(* IEC 61131-3 sources: industrial-ai-agent/projects/EXAMPLE_conveyor/program, 4 files *)

(* ---- 00_DUTs.st ---- *)
// ============================================================
// DUT (Data Unit Types) — Numaralandirmalar
// Proje: EXAMPLE_Conveyor_Line1
// Aciklama: Bolge mod ve durum makinesi tipleri
// ============================================================

// Bolge calisma modu
TYPE E_ZoneMode :
(
    MODE_MANUAL := 0,   // Operator buton ile kontrol
    MODE_AUTO   := 1    // Otomatik sira / fotosel ile
) := MODE_MANUAL;
END_TYPE

// Bolge durum makinesi
TYPE E_ZoneState :
(
    STATE_IDLE     := 0,    // Bekliyor, motor kapali
    STATE_STARTING := 1,    // Baslatma gecisi
    STATE_RUNNING  := 2,    // Calisiyor
    STATE_STOPPING := 3,    // Durdurma gecisi
    STATE_JAMMED   := 4,    // Sikisma - reset bekliyor
    STATE_FAULT    := 5     // Hata (hiz/diger) - reset bekliyor
) := STATE_IDLE;
END_TYPE

(* ---- 01_GVL_IO.st ---- *)
// ============================================================
// GVL_IO — Fiziksel Giris/Cikis degiskenleri
// Adresler io_list.csv ile BIREBIR tutarli olmalidir.
// Tek-yazar disiplini: cikislari yalniz ilgili PRG yazar.
// ============================================================
{attribute 'qualified_only'}
VAR_GLOBAL
    // --- Dijital Girisler (DI) ---
    ZN1_SEL_01_Auto    AT %IX0.0 : BOOL;   // Bolge 1 Oto/Manuel
    ZN1_PBS_01_Start   AT %IX0.1 : BOOL;
    ZN1_PBS_01_Stop    AT %IX0.2 : BOOL;   // NC: 1=normal, 0=basili
    ZN1_JAM_01_Sensor  AT %IX0.3 : BOOL;
    ZN1_PEY_01_Present AT %IX0.4 : BOOL;
    ZN2_SEL_02_Auto    AT %IX0.5 : BOOL;
    ZN2_PBS_02_Start   AT %IX0.6 : BOOL;
    ZN2_PBS_02_Stop    AT %IX0.7 : BOOL;
    ZN2_JAM_02_Sensor  AT %IX1.0 : BOOL;
    ZN2_PEY_02_Present AT %IX1.1 : BOOL;
    ZN3_SEL_03_Auto    AT %IX1.2 : BOOL;
    ZN3_PBS_03_Start   AT %IX1.3 : BOOL;
    ZN3_PBS_03_Stop    AT %IX1.4 : BOOL;
    ZN3_JAM_03_Sensor  AT %IX1.5 : BOOL;
    ZN3_PEY_03_Present AT %IX1.6 : BOOL;
    PLT_EST_01_OK      AT %IX1.7 : BOOL;   // Acil durdurma zinciri saglam (NC=1)
    PLT_RST_01_PB      AT %IX2.0 : BOOL;   // Reset / hata kabul
    PLT_PMT_01_Run     AT %IX2.1 : BOOL;   // Calistirma izni (NC)

    // --- Dijital Cikislar (DO) ---
    ZN1_MTR_01_Run     AT %QX0.0 : BOOL;
    ZN1_LMP_01_Run     AT %QX0.1 : BOOL;
    ZN1_LMP_01_Flt     AT %QX0.2 : BOOL;
    ZN2_MTR_02_Run     AT %QX0.3 : BOOL;
    ZN2_LMP_02_Run     AT %QX0.4 : BOOL;
    ZN2_LMP_02_Flt     AT %QX0.5 : BOOL;
    ZN3_MTR_03_Run     AT %QX0.6 : BOOL;
    ZN3_LMP_03_Run     AT %QX0.7 : BOOL;
    ZN3_LMP_03_Flt     AT %QX1.0 : BOOL;
    PLT_BCN_01_Run     AT %QX1.1 : BOOL;
    PLT_BCN_01_Flt     AT %QX1.2 : BOOL;
    PLT_HRN_01_Alarm   AT %QX1.3 : BOOL;

    // --- Analog Girisler (AI) — 4-20mA takometre ---
    ZN1_TAC_01_Speed   AT %IW2 : INT;
    ZN2_TAC_02_Speed   AT %IW3 : INT;
    ZN3_TAC_03_Speed   AT %IW4 : INT;
END_VAR

(* ---- 02_GVL_Const_HMI.st ---- *)
// ============================================================
// GVL_Const — Sabitler (sihirli sayi yok kurali)
// ============================================================
{attribute 'qualified_only'}
VAR_GLOBAL CONSTANT
    // Analog olcekleme (4-20mA, modul ham deger araligi varsayimi 0..32767)
    RAW_4MA      : INT  := 6553;     // 4mA  -> ham deger (~%20)
    RAW_20MA     : INT  := 32767;    // 20mA -> ham deger (tam skala)
    RAW_BREAK    : INT  := 3276;     // <2mA -> kablo kopmasi esigi (NAMUR NE107)
    SPEED_ENG_MIN: REAL := 0.0;      // m/min
    SPEED_ENG_MAX: REAL := 120.0;    // m/min

    // Hiz arizasi tespiti
    SPEED_MIN_RUN  : REAL := 5.0;          // Calisirken beklenen min hiz (m/min)
    T_SPEED_CHECK  : TIME := T#2S;         // Hiz kontrol gecikmesi

    // Zamanlamalar
    T_JAM_DEBOUNCE : TIME := T#200MS;      // Sikisma debounce (spec)
    T_START_RAMP   : TIME := T#500MS;      // Baslatma gecis suresi
    T_STOP_RAMP    : TIME := T#300MS;      // Durdurma gecis suresi
END_VAR

// ============================================================
// GVL_HMI — OPC-UA / HMI'a acilan degiskenler
// Bu degiskenler Symbol Configuration ile OPC-UA node olur.
// HMI yalniz OPC-UA uzerinden okur; kontrol mantigi HMI'da DEGIL.
// Komutlar (xCmd*) HMI'dan yazilir; geri kalan salt-okunur izlemedir.
// ============================================================
{attribute 'qualified_only'}
VAR_GLOBAL
    // Izleme (PLC -> HMI, salt okunur)
    aZoneState   : ARRAY[1..3] OF E_ZoneState;   // Bolge durumlari
    aZoneSpeed   : ARRAY[1..3] OF REAL;          // m/min
    aZoneRunning : ARRAY[1..3] OF BOOL;
    aZoneJam     : ARRAY[1..3] OF BOOL;
    aZoneSpdFlt  : ARRAY[1..3] OF BOOL;
    aZoneTacBrk  : ARRAY[1..3] OF BOOL;           // Takometre kablo kopmasi
    aZoneAuto    : ARRAY[1..3] OF BOOL;
    xEStopActive : BOOL;                          // A001
    xRunPermit   : BOOL;                          // PLT_PMT durumu
    xZone2Itlk   : BOOL;                          // A060 interlock blokaji
    xAnyAlarm    : BOOL;

    // Komut (HMI -> PLC) — yalniz OTO modda gecerli, manuelde butonlar onceliklidir
    axCmdAutoRun : ARRAY[1..3] OF BOOL;           // Oto mod calistirma istegi
    xCmdReset    : BOOL;                          // HMI'dan reset (PLT_RST ile OR'lanir)

    // Heartbeat — HMI baglanti kopmasini tespit eder (her saniye toggle)
    uHeartbeat   : UDINT;
END_VAR

(* ---- 03_FB_AnalogScale.st ---- *)
// ============================================================
// FB_AnalogScale
// Aciklama: 4-20mA ham analog degeri muhendislik birimine
//           cevirir. Kablo kopmasi (under-range, NAMUR NE107)
//           ve over-range tespiti yapar. Tek sorumluluk: olcekleme.
// ============================================================
FUNCTION_BLOCK FB_AnalogScale
VAR_INPUT
    iRaw     : INT;    // Modulden gelen ham deger
    iRawMin  : INT;    // 4mA karsiligi ham deger
    iRawMax  : INT;    // 20mA karsiligi ham deger
    rEngMin  : REAL;   // Muhendislik min
    rEngMax  : REAL;   // Muhendislik max
    iRawBreak: INT;    // Altinda kablo kopmasi sayilan esik
END_VAR
VAR_OUTPUT
    rEng       : REAL;   // Olceklenmis deger
    xUnderRange: BOOL;   // Kablo kopmasi / 4mA alti
    xOverRange : BOOL;   // 20mA ustu
END_VAR
VAR
    rSpan : REAL;
END_VAR

// --- Kablo kopmasi kontrolu (once) ---
xUnderRange := (iRaw < iRawBreak);

IF xUnderRange THEN
    rEng := rEngMin;        // Guvenli varsayilan: min deger
    xOverRange := FALSE;
    RETURN;
END_IF

// --- Sifira bolme korumasi ---
rSpan := INT_TO_REAL(iRawMax - iRawMin);
IF rSpan <= 0.0 THEN
    rEng := rEngMin;        // Hatali konfig - guvenli deger
    RETURN;
END_IF

// --- Lineer olcekleme ---
rEng := rEngMin + (INT_TO_REAL(iRaw - iRawMin) / rSpan) * (rEngMax - rEngMin);

// --- Kelepceleme (clamp) ---
xOverRange := (rEng > rEngMax);
IF rEng > rEngMax THEN
    rEng := rEngMax;
ELSIF rEng < rEngMin THEN
    rEng := rEngMin;
END_IF
